// TIA Portal V18 export
VAR_GLOBAL   // PLC tag table "IV3"
END_VAR
VAR_GLOBAL CONSTANT   // user constants
   MS_MANUAL : Int := 1;
   MS_EMPTY : Int := 0;
   MS_Auto : Int := 2;
END_VAR
